TYPE ST_WinchParameters :
STRUCT
	fEncoderOffset : LREAL := 17574.8;
	fWinchDrumScaling : LREAL := 0.000744309;
	fWinchMotorDisplacement : LREAL := 32.0; 
	fWinchMaxSpeed : LREAL := 0.05; // rad/s
	
END_STRUCT
END_TYPE

(* stored: Version 1.1.0.1, ProductVersion 3.1.4024.12
   DUT ST_WinchParameters: Id {5715d113-58b0-4176-b35d-152e541ba749} *)
